Fanuc KAREL source: ka00119.KL

PROGRAM KA00119
%STACKSIZE=65535
%PRIORITY=65535
%NOLOCKGROUP
-- UNRESOLVED DECLARATIONS (source type spelling not recovered)
-- SRC : TYPE_0x001C (type_u16=0x001C)
-- DST : ARRAY[2] OF TYPE_0x0018 (type_u16=0x2018)
BEGIN
-- UNRESOLVED_PC line 7 opcodes [9D 22 A5] marker_code=0
DST[1]=SRC
END KA00119
